{attribute 'qualified_only'}
{attribute 'strict'}
TYPE E_LED_MODES :
(
    SOLID_YELLOW := 0,
    FLASH_YELLOW := 1,
    SOLID_RED := 2,
    FLASH_RED := 3,
    SOLID_GREEN := 4
);
END_TYPE

(* stored: Version 1.1.0.1, ProductVersion 3.1.4024.11
   DUT E_LED_MODES: Id {86f86d08-88f0-44ab-bd2a-e10eac74146c} *)
